PROGRAM prgHouse
VAR
	fbHouse				: FB_HouseC_Power_Virtual;
	bHouseEnabled		: BOOL;						//{#lynus.ag#()}
	lrPowerHouse		: LREAL;					//{#lynus.ag#()}
	lrPowerHouse_Manual	: LREAL;					//{#lynus.ag#()}
	lrPowerHouseUndelayed: LREAL;					//{#lynus.ag#()}
END_VAR
VAR PERSISTENT
	bEnableHouse		: BOOL;						//{#lynus.ag#()}
END_VAR

fbHouse(
	bEnable:= bEnableHouse, 
	diNrOfEMS_IN:= prgEMS.fbEMS.diNrOfEMS_OUT, 
	bSetDefault:= , 
	lrCounterConsumptionSetDefault:= , 
	lrCounterProductionSetDefault:= , 
	stDataHouseC=> , 
	diNrOfHouseC_OUT=> );
	
bHouseEnabled := fbHouse.stDataHouseC.bEnabled;
// lrPowerHouse := fbHouse.stDataHouseC.lrPower; 		// not calculating correctly	
lrPowerHouse_Manual := prgPV.lrPowerPV + prgGrid.lrPowerGrid;

lrPowerHouse:= MAX(0,lrPowerHouse_Manual)- prgTemperature.real_PowerHeater;
lrPowerHouseUndelayed := prgGrid.fbEM1.stDataEMPowerRealTime.lrPowerTotal + prgPV.lrPowerPV - prgTemperature.real_PowerHeater;

END_PROGRAM

(* stored: Version 1.1.0.1, ProductVersion 3.1.4024.12
   POU prgHouse: Id {1004e12f-88fd-4838-a3c1-f7a079c901cf}, SpecialFunc None *)
